TYPE ST_System_Events :
STRUCT
	b_RestartRequiredMachineName		: BOOL;
	b_TimeUpdateFailed					: BOOL;
END_STRUCT
END_TYPE

(* stored: Version 1.1.0.1, ProductVersion 3.1.4026.18
   DUT ST_System_Events: Id {a049eaed-f5ed-42a5-958f-42e53da2979e} *)
